{attribute 'GeneratedUsingTerminal: EL6784-0000-0016'}
{attribute addProperty BoxType "EL6784-0000-0016"}
{attribute addProperty Id "StatusAT %I*Status_07D3AAF62InputsEMPTY_STRUCTURE0ControlAT %Q*Control_DAFD38E02OutputsEMPTY_STRUCTURE0WcStateAT %I*WcState_9091E0EB2InfoDataAT %I*InfoData_32EB74EA10"}
{attribute addProperty CRC "2640427583"}
{attribute addProperty Size "16"}
TYPE EL6784_9D61BA3F EXTENDS EtcSlaveTerminalBase_947E5A46 :
STRUCT
	{attribute addProperty Name "Status"}
	Status : Status_07D3AAF6;
	{attribute addProperty Name "Inputs"}
	Inputs : EMPTY_STRUCTURE;
	{attribute addProperty Name "Control"}
	Control : Control_DAFD38E0;
	{attribute addProperty Name "Outputs"}
	Outputs : EMPTY_STRUCTURE;
	{attribute addProperty Name "WcState"}
	WcState : WcState_9091E0EB;
	{attribute addProperty Name "InfoData"}
	InfoData : InfoData_32EB74EA;
END_STRUCT
END_TYPE

(* stored: Version 1.2.0.0, ProductVersion 3.1.4024.9
   DUT EL6784_9D61BA3F: Id {37377d64-78bf-4594-87b7-e84c6552c847} *)
